// TwinCAT 3 PLC project hxx_vonhamos
// ProgramVersion: 3.1.4022.7
// libraries:
//   Tc2_Standard, * (Beckhoff Automation GmbH)
//   Tc2_System, * (Beckhoff Automation GmbH)
//   Tc3_Module, * (Beckhoff Automation GmbH)
//   lcls-twincat-motion,1.3.2,SLAC
// project tree:
//   / PlcTask.TcTTO (not stored)
//   POUs/ Main.TcPOU
// real-time tasks:
//   TASK PlcTask: cycle T#10ms, priority 20, ADS port 350
// motion (NC):
// I/O:
//   DEVICE Device 1 (EtherCAT), AmsNetId 5.63.55.4.2.1
//     VonHamos_EK1200_E0
// variable links:
//   hxx_vonhamos Instance <-> Device 1 (EtherCAT)/VonHamos_EK1200_E0/VonHamos_EL1084_E2
//     PlcTask Inputs/Main.M1.bHome <-> Channel 3/Input
//     PlcTask Inputs/Main.M1.bLimitBackwardEnable <-> Channel 2/Input
//     PlcTask Inputs/Main.M1.bLimitForwardEnable <-> Channel 1/Input
//   hxx_vonhamos Instance <-> Device 1 (EtherCAT)/VonHamos_EK1200_E0/VonHamos_EL2004_E7
//     PlcTask Outputs/Main.M1.bBrakeRelease <-> Channel 1/Output
//   hxx_vonhamos Instance <-> NC-Task 1 SAF/Axes/VonHamosY
//     PlcTask Inputs/Main.M1.Axis.NcToPlc <-> Outputs/ToPlc
//     PlcTask Outputs/Main.M1.Axis.PlcToNc <-> Inputs/FromPlc

// ---- POUs/Main.TcPOU
PROGRAM Main
VAR
	// Motors
	{attribute 'TcLinkTo' := '.bLimitForwardEnable	:=TIIB[VonHamos_EL1084_E2]^Channel 1^Input;
                              .bLimitBackwardEnable	:=TIIB[VonHamos_EL1084_E2]^Channel 2^Input;
							  .bHome				:=TIIB[VonHamos_EL1084_E2]^Channel 3^Input;
							  .bBrakeRelease		:=TIIB[VonHamos_EL2004_E7]^Channel 1^Output'}
	{attribute 'pytmc' := '
		pv: HXX:VON_HAMOS:MMS:01
	'}
	M1 : DUT_MotionStage; // Y axis

	fbMotionStageM1 : FB_MotionStage;
END_VAR

// Hardware Enable
M1.bPowerSelf := TRUE;
M1.bHardwareEnable := TRUE;
fbMotionStageM1(stMotionStage:=M1);

END_PROGRAM
